PROGRAM prgLab10_11
VAR
	motor:FB_Motor;
	bLiga AT %I*: BOOL;
	bDesliga AT %I*: BOOL;
	reset AT %I*: BOOL;
	temperatura: REAL;
	saidaMotor AT %Q*: BOOL;
	error AT %Q*: BOOL;
	analogInput AT %I*: INT;
END_VAR

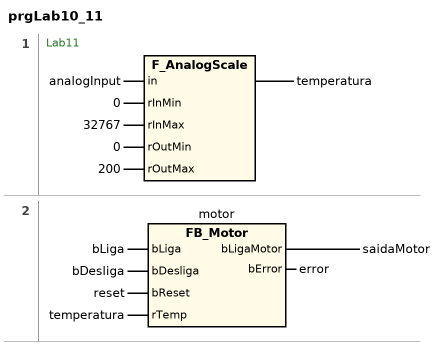
// NETWORK 1
// Lab11
temperatura := F_AnalogScale(in := analogInput, rInMin := 0, rInMax := 32767, rOutMin := 0, rOutMax := 200);

// NETWORK 2
motor(bLiga := bLiga, bDesliga := bDesliga, bReset := reset, rTemp := temperatura, bError => error); // FB_Motor
saidaMotor := motor.bLigaMotor;

END_PROGRAM

(* stored: Version 1.1.0.1, ProductVersion 3.1.4024.11
   POU prgLab10_11: Id {38ca7319-d331-4814-8755-a931249efa42}, SpecialFunc None *)
